FUNCTION_BLOCK FB_TOR_DS EXTENDS FB_TOR_Base
//////////////////
//  Door sensor system . State = True >> Door Closed .
//////////////////

VAR_INPUT PERSISTENT
	// Parameters of the Object (instance/model specific) 
		ParamTempoDoorAlarm			: TIME := T#10S ;	(* (s) Tempo for Door sensor alarm *)
		
END_VAR

VAR_OUTPUT
	//Child objects
	
END_VAR

VAR_INPUT
	// I/O Inputs 		                                     				
	MesDataExd			: TOR_Standard ;  
		
END_VAR

VAR
	//M_ALARMMANAGEMENT VARIABLES//
		TON_Ouverture				: TON;				//(NA) Tempo to detect door opened for too long time . 



END_VAR

METHOD M_AlarmManagement
//////////////////
// Manages Door sensor alarms and warnings
/////////////////

VAR 
	// Method local variables (reinitialized at each cycle) 
	FB_AlarmCodeManager : FB_AlarmCodeManager ; 


END_VAR
// Detection Variables
TON_Ouverture(IN:= MesDataExd.MesData.MesAlarmState,PT:=ParamTempoDoorAlarm);

// ALARM CODE //
	FB_AlarmCodeManager(
 		bAlarm1			:= FALSE,    	// 
		bAlarm2			:= FALSE, 		// 
		bAlarm3			:= FALSE, 		// 
		bAlarm4			:= FALSE, 		// 
		bAlarm5			:= FALSE,       //
		bAlarm6			:= FALSE,       //
		bAlarm7			:= FALSE,       //
		bAlarm8			:= FALSE,       //
		bAlarm9			:= FALSE,       //
		bAlarm10		:= FALSE,       //
		bAlarm11		:= FALSE,       //
		bAlarm12		:= FALSE,       //
		bAlarm13		:= FALSE,       //
		bAlarm14		:= FALSE,       //
		bAlarm15		:= FALSE,       //
		wAlarmCode		=>MesDataExd.MesData.MesAlarmCode);

// WARNING CODE //
	FB_AlarmCodeManager(
		bAlarm1			:= TON_Ouverture.Q,    	// The door is opened for more than 15 seconds
		bAlarm2			:= FALSE, 				// 
		bAlarm3			:= FALSE, 				// 
		bAlarm4			:= FALSE, 				// 
		bAlarm5			:= FALSE, 				//
		bAlarm6			:= FALSE,               //
		bAlarm7			:= FALSE,               //
		bAlarm8			:= FALSE,               //
		bAlarm9			:= FALSE,               //
		bAlarm10		:= FALSE,               //
		bAlarm11		:= FALSE,               //
		bAlarm12		:= FALSE,               //
		bAlarm13		:= FALSE,               //
		bAlarm14		:= FALSE,               //
		bAlarm15		:= FALSE,               //
		wAlarmCode		=>MesDataExd.MesData.MesWarningCode);

// EVENT CODE //
	FB_AlarmCodeManager(
		bAlarm1			:= MesDataExd.MesData.MesAlarmState, 		// Door is Opened
		bAlarm2			:= FALSE, 						// 
		bAlarm3			:= FALSE, 						// 
		bAlarm4			:= FALSE, 						// 
		bAlarm5			:= FALSE, 						//
		bAlarm6			:= FALSE, 						//
		bAlarm7			:= FALSE, 						//
		bAlarm8			:= FALSE, 						//
		bAlarm9			:= FALSE, 						//
		bAlarm10		:= FALSE, 						//
		bAlarm11		:= FALSE, 						//
		bAlarm12		:= FALSE, 						//
		bAlarm13		:= FALSE, 						//
		bAlarm14		:= FALSE, 						//
		bAlarm15		:= FALSE, 						//
		wAlarmCode		=>MesDataExd.MesData.MesEventCode);
END_METHOD

METHOD M_Execute
//////////////////
//  Method Calls 
/////////////////

VAR 
	// Method local variables (reinitialized at each cycle) 
	
END_VAR


SUPER^.M_Execute() ;
END_METHOD

METHOD M_StateManager
//////////////////
// Detect when fire occurs
/////////////////

VAR 
	// Method local variables (reinitialized at each cycle)
 	MesStateInterm1 : BOOL;
	MesStateInterm2 : BOOL;
END_VAR

IF ParamCableCutSecurity THEN
	MesStateInterm1 := NOT IN_MesState1_IO ; 
	MesStateInterm2 := NOT IN_MesState2_IO ; 
ELSE 
	MesStateInterm1 := IN_MesState1_IO;
	MesStateInterm2 := IN_MesState2_IO;
END_IF

IF ParamNbSensors = 1 THEN 
	MesStateInterm2 := MesStateInterm1 ;
END_IF

IF ParamAtleastOne THEN 
MesDataExd.MesData.MesAlarmState := MesStateInterm1 OR MesStateInterm2 ; 
ELSE
MesDataExd.MesData.MesAlarmState := MesStateInterm1 AND MesStateInterm2 ; 
END_IF

R_TRIGAlarm(CLK:= MesDataExd.MesData.MesAlarmState ) ; 
IF R_TRIGAlarm.Q THEN
	MesCountAlarm :=  MIN(MesCountAlarm + 1 ,4294967295 ) ; 
ELSIF IN_ResetCounter THEN 
	MesCountAlarm := 0 ; 
END_IF

MesDataExd.MesData.MesCountAlarm	:= MesCountAlarm ;
END_METHOD

END_FUNCTION_BLOCK

(* stored: Version 1.1.0.1, ProductVersion 3.1.4024.12
   POU FB_TOR_DS: Id {3296ffca-bfc4-4222-8531-79e922ab77c0}, SpecialFunc None
   Method M_AlarmManagement: Id {c8bf3d3b-9cbc-4386-b814-4514b9e39e02}
   Method M_Execute: Id {0ad2967f-5ee3-469a-92ac-3a04f973cd7a}
   Method M_StateManager: Id {c3775f9f-eaaf-48de-9fb6-e609b14bf74b} *)
